ABB RobotStudio station: test1.rsstn

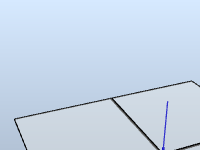
Station test1 (saved by RobotStudio 6.8.8148.134)
Layout (positions relative to the parent item):
